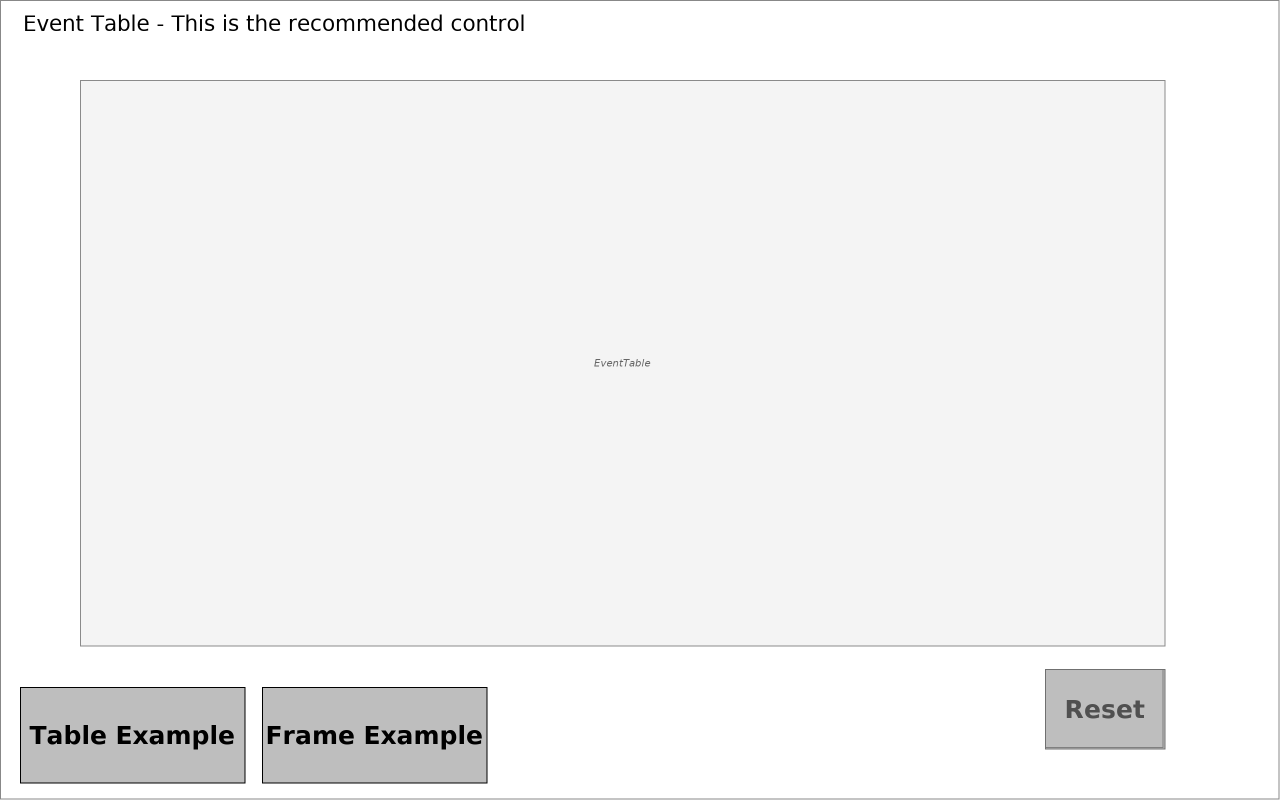
VISUALIZATION Event_Table  // 1280x800
    Rectangle (20,9 909x60), "Event Table - This is the recommended control"
    Rectangle (20,687 225x96), "Table Example"
        OnMouseClick: change screen: Alarm_Table
    EventTable (80,80 1085x566)
        p1690906150: Class
        p3258520714: Date
        p2231227367: Time
        p3993844394: Message
        p2076579579: Details
        p3558512729: MAIN.fbReadEvents.aEvents
        p3921149237: m_pDataArray..pArray
    Button (1045,669 120x80), "Reset"
        tap HMI.xFaultResetPB
    Rectangle (262,687 225x96), "Frame Example"
        OnMouseClick: change screen: Alarms
END_VISUALIZATION

(* stored: Version 1.1.0.1
   Visu Event_Table: Id {58fed1c3-5634-4f1b-8a3a-9cc1774acb69} *)
